TYPE ST_Config_Valve:
STRUCT
END_STRUCT
END_TYPE

(* stored: Version 1.1.0.1, ProductVersion 3.1.4019.2
   DUT ST_Config_Valve: Id {1e5eceea-3093-4235-b042-7f427d397e5f} *)
